TYPE ST_GC_Signal_Out :
STRUCT
	bVaccumOn : BOOL;

	bDOs : ARRAY[1..16] OF BOOL;
	rAOs : ARRAY[1..16] OF REAL;
END_STRUCT
END_TYPE

(* stored: Version 1.1.0.1, ProductVersion 3.1.4026.18
   DUT ST_GC_Signal_Out: Id {9921dc3d-b38f-43b3-84f6-12803bd60c4e} *)
